(* IEC 61131-3 sources: teller/JD_Teller_LC2_V11/Class/ChannelBaseDataWriteOnly, 1 file *)

(* ---- ChannelBaseDataWriteOnly.st ---- *)
(*!
<Class
	Name               = "ChannelBaseDataWriteOnly"
	Revision           = "1.0"
	RealtimeTask       = "false"
	CyclicTask         = "false"
	BackgroundTask     = "false"
	Sigmatek           = "true"
	OSInterface        = "false"
	HighPriority       = "false"
	Automatic          = "false"
	UpdateMode         = "Prescan"
	IconPath           = ".\Class\Tool.ico"
	SharedCommandTable = "true"
	Objectsize         = "(284,120)">
	<Channels>
	</Channels>
	<RevDoku>
		<Owner Company="Sigmatek" Author="BleErn"/>
		<Dokumentation Revision="1.0" Date="04.03.2010" Author="BleErn" Company="Sigmatek" Description="New Base Class for Input/Output-Channel-Classes"/>
	</RevDoku>
	<Network Name="ChannelBaseDataWriteOnly">
		<!-- List of Components in this network -->
		<Components>
			<Object
				Name       = "_base"
				Class      = "ChannelBaseData"
				Position   = "(218,120)"
				Visualized = "false">
				<Channels>
					<Server Name="Data"/>
				</Channels>
			</Object>
		</Components>
		<Comments>
		</Comments>
		<!-- List of Connections in this network -->
		<Connections>
			<Connection Source="this.Data" Destination="_base.Data" Vertices="(690,210),(518,210),"/>
		</Connections>
		<!-- Headerfiles -->
		<Options>
		</Options>
	</Network>
</Class>
*)
#pragma using ChannelBaseData

ChannelBaseDataWriteOnly : CLASS
: ChannelBaseData
  //Servers:
  //Clients:
  //Variables:
  //Functions:

	FUNCTION VIRTUAL GLOBAL UpDateRt
		VAR_INPUT
			Handle 	: DINT;
		END_VAR;
  //Tables:
	FUNCTION @STD
		VAR_OUTPUT
			ret_code	: CONFSTATES;
		END_VAR;
	FUNCTION GLOBAL TAB @CT_;
END_CLASS;

#pragma warning(disable: 73 )
FUNCTION VIRTUAL GLOBAL ChannelBaseDataWriteOnly::UpDateRt
	VAR_INPUT
		Handle 	: DINT;
	END_VAR

END_FUNCTION
#pragma warning(default: 73 )
